// TIA Portal V20 export
TYPE "LCFL_typeMTPMonBinVlvSiemens"
TITLE = MTP for monitoring binary valve (Siemens) / MTP für binäre Ventilüberwachung (Siemens)
// MTP data for bistable valve with the feedback monitoring (Siemens) / MTP-Daten für bistabiles Ventil mit Rückmeldeüberwachung (Siemens)
   STRUCT
      mtpData : "LCFL_typeMTPMonBinVlv";
      maintenance : "LCFL_typeMaintenance";
      tagName { ExternalWritable := 'False'} : String[30] := '';   // Instanznamen-Identifizierung / Instance name identification
      enabled { ExternalWritable := 'False'} : Bool := FALSE;   // Funktionalität des Steuerelements ist aktiviert / Functionality of control module is enabled
      monitorStaticMessage { ExternalWritable := 'False'} : Bool := FALSE;   // Meldung für statischen Fehler (1: Meldung ist aktiviert; 0: Meldung ist deaktiviert) / Message for static error (1: Message active; 0: Message inactive)
      monitorDynamicMessage { ExternalWritable := 'False'} : Bool := FALSE;   // Meldung für dynamischen Fehler (1: Meldung ist aktiviert; 0: Meldung ist deaktiviert) / Message for dynamic error (1: Message active; 0: Message inactive)
      operatingTimeMessage { ExternalWritable := 'False'} : Bool := FALSE;   // Meldung für Betriebsstunden haben ihre Grenze erreicht (1: Meldung ist aktiviert; 0: Meldung ist deaktiviert) / Message for operating time has reached (1: Message active; 0: Message inactive)
      cycleTimeMessage { ExternalWritable := 'False'} : Bool := FALSE;   // Meldung für Zykluszeit ist erreicht (1: Meldung aktiv; 0: Meldung inaktiv) / Message for cycle time has reached (1: Message active; 0: Message inactive)
      switchCounterMessage { ExternalWritable := 'False'} : Bool := FALSE;   // Meldung für Anzahl der Zustandswechsel hat seine Grenze erreicht (1: Meldung ist aktiviert; 0: Meldung ist deaktiviert) / Message for switch counter has reached (1: Message active; 0: Message inactive)
      alarmCounterMessage { ExternalWritable := 'False'} : Bool := FALSE;   // Meldung für Alarmzähler ist erreicht (1: Meldung aktiv; 0: Meldung inaktiv) / Message for alarm counter has reached (1: Message active; 0: Message inactive)
      interconnectorActive { ExternalWritable := 'False'} : Bool := FALSE;   // Interconnector active (1: Active; 0: Inactive)
      interconnectedTagName { ExternalWritable := 'False'} : String[30] := '';   // Name der verbundenen Instanz / Name of interconnected instance
   END_STRUCT;
END_TYPE
